SUBAPPLICATION Uebung_HystereseVertikal_AX_simple (* MID/DEAD/HYSTERESIS-Eingabefelder bewegen live die 5 Schwellwert-Dreiecke im vertikalen Bargraph (Type=1 BottomToTop, Pixelposition gespiegelt: hoher Wert = kleiner Top) *)
  (* Standard: 61499-2; Description: Copyright (c) 2026 Meisterschulen am Ostbahnhof This program and the accompanying materials are made available under the terms of the Eclipse Public License 2.0 which is available at https://www.eclipse.org/legal/epl-2.0/ SPDX-License-Identifier: EPL-2.0 *)
  (* Version 1.2, 2026-09-27, Franz Höpfinger, Meisterschulen am Ostbahnhof, Schwellwert-Berechnung zu MyLib::sys::DualHysteresis_Thresholds_AR ausgelagert *)
  (* Version 1.1, 2026-09-27, Franz Höpfinger, Meisterschulen am Ostbahnhof, AR_TO_AI, Zero, QPos zu MyLib::sys::Q_ChildPosition_AR_Vertikal SubApp ausgelagert *)
  PACKAGE Uebungen;
  IMPORT Uebungen::const::UT::HystereseVertikal::DefaultPool_Numeric::InputNumber_MID_N;
  IMPORT Uebungen::const::UT::HystereseVertikal::DefaultPool_Numeric::InputNumber_DEAD_N;
  IMPORT Uebungen::const::UT::HystereseVertikal::DefaultPool_Numeric::InputNumber_HYSTERESIS_N;
  IMPORT Uebungen::const::UT::HystereseVertikal::DefaultPool::Polygon_MID;
  IMPORT Uebungen::const::UT::HystereseVertikal::DefaultPool::Polygon_MID_PLUS_DEAD;
  IMPORT Uebungen::const::UT::HystereseVertikal::DefaultPool::Polygon_MID_MINUS_DEAD;
  IMPORT Uebungen::const::UT::HystereseVertikal::DefaultPool::Polygon_MID_PLUS_DEAD_HYST;
  IMPORT Uebungen::const::UT::HystereseVertikal::DefaultPool::Polygon_MID_MINUS_DEAD_HYST;
  IMPORT Uebungen::const::UT::HystereseVertikal::DefaultPool::Container_Schwellwerte;
  IMPORT Uebungen::const::UT::HystereseVertikal::DefaultPool_Bargraph::Bargraph_Hysterese_ScalePx;
  IMPORT Uebungen::const::UT::HystereseVertikal::DefaultPool_Bargraph::Bargraph_Hysterese_LengthPx;
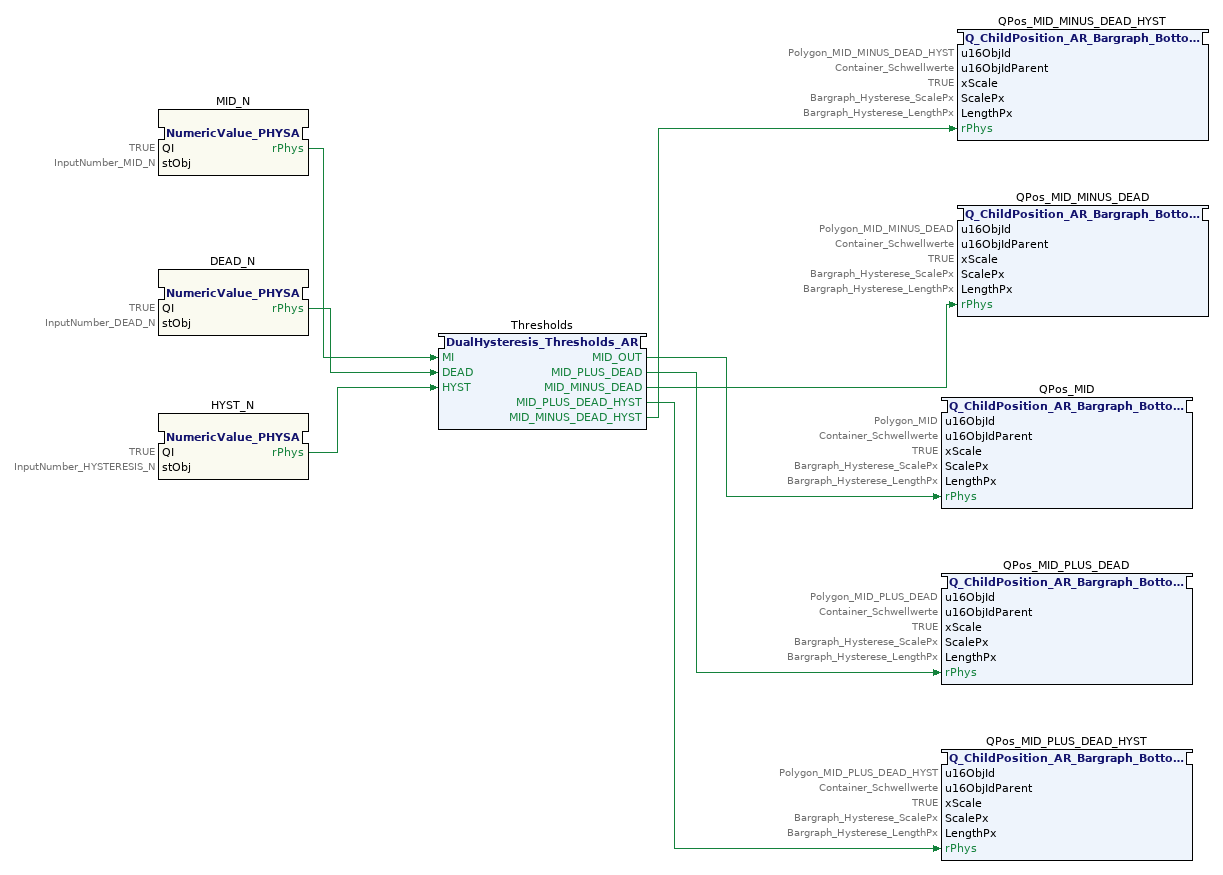
  FBS
    MID_N : isobus::UT::io::NumericValue::NumericValue_PHYSA(QI := TRUE, stObj := InputNumber_MID_N);
    DEAD_N : isobus::UT::io::NumericValue::NumericValue_PHYSA(QI := TRUE, stObj := InputNumber_DEAD_N);
    HYST_N : isobus::UT::io::NumericValue::NumericValue_PHYSA(QI := TRUE, stObj := InputNumber_HYSTERESIS_N);
  END_FBS
  SUBAPPS
    Thresholds : MyLib::sys::DualHysteresis_Thresholds_AR;
    QPos_MID : MyLib::sys::Q_ChildPosition_AR_Bargraph_BottomToTop(u16ObjId := Polygon_MID, u16ObjIdParent := Container_Schwellwerte, xScale := TRUE, ScalePx := Bargraph_Hysterese_ScalePx, LengthPx := Bargraph_Hysterese_LengthPx);
    QPos_MID_PLUS_DEAD : MyLib::sys::Q_ChildPosition_AR_Bargraph_BottomToTop(u16ObjId := Polygon_MID_PLUS_DEAD, u16ObjIdParent := Container_Schwellwerte, xScale := TRUE, ScalePx := Bargraph_Hysterese_ScalePx, LengthPx := Bargraph_Hysterese_LengthPx);
    QPos_MID_MINUS_DEAD : MyLib::sys::Q_ChildPosition_AR_Bargraph_BottomToTop(u16ObjId := Polygon_MID_MINUS_DEAD, u16ObjIdParent := Container_Schwellwerte, xScale := TRUE, ScalePx := Bargraph_Hysterese_ScalePx, LengthPx := Bargraph_Hysterese_LengthPx);
    QPos_MID_PLUS_DEAD_HYST : MyLib::sys::Q_ChildPosition_AR_Bargraph_BottomToTop(u16ObjId := Polygon_MID_PLUS_DEAD_HYST, u16ObjIdParent := Container_Schwellwerte, xScale := TRUE, ScalePx := Bargraph_Hysterese_ScalePx, LengthPx := Bargraph_Hysterese_LengthPx);
    QPos_MID_MINUS_DEAD_HYST : MyLib::sys::Q_ChildPosition_AR_Bargraph_BottomToTop(u16ObjId := Polygon_MID_MINUS_DEAD_HYST, u16ObjIdParent := Container_Schwellwerte, xScale := TRUE, ScalePx := Bargraph_Hysterese_ScalePx, LengthPx := Bargraph_Hysterese_LengthPx);
  END_SUBAPPS
  ADAPTER_CONNECTIONS
    MID_N.rPhys TO Thresholds.MI;
    DEAD_N.rPhys TO Thresholds.DEAD;
    HYST_N.rPhys TO Thresholds.HYST;
    Thresholds.MID_OUT TO QPos_MID.rPhys;
    Thresholds.MID_PLUS_DEAD TO QPos_MID_PLUS_DEAD.rPhys;
    Thresholds.MID_MINUS_DEAD TO QPos_MID_MINUS_DEAD.rPhys;
    Thresholds.MID_PLUS_DEAD_HYST TO QPos_MID_PLUS_DEAD_HYST.rPhys;
    Thresholds.MID_MINUS_DEAD_HYST TO QPos_MID_MINUS_DEAD_HYST.rPhys;
  END_CONNECTIONS
END_SUBAPPLICATION
